// Mitsubishi GX Works2 project: plc   PLC: Q06UDV

PROGRAM MAIN
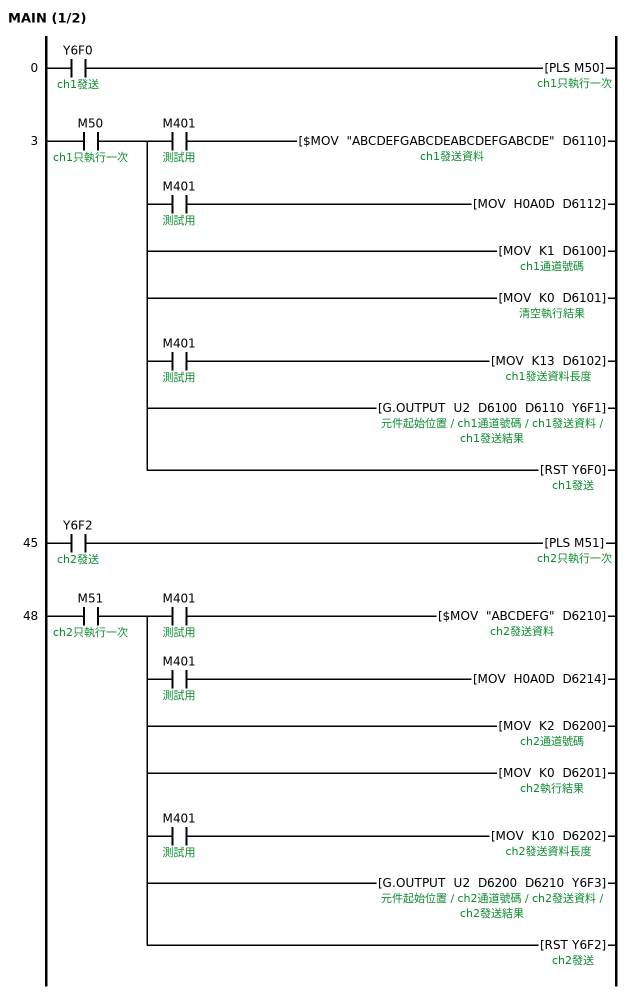
0     LD      Y6F0  ; ch1發送
      PLS     M50  ; ch1只執行一次
3     LD      M50  ; ch1只執行一次
      MPS
      AND     M401  ; 測試用
      $MOV    "ABCDEFGABCDEABCDEFGABCDE" D6110  ; ch1發送資料
      MRD
      AND     M401  ; 測試用
      MOV     H0A0D D6112
      MPP
      MOV     K1 D6100  ; ch1通道號碼
      MOV     K0 D6101  ; 清空執行結果
      MPS
      AND     M401  ; 測試用
      MOV     K13 D6102  ; ch1發送資料長度
      MPP
      G.OUTPUT U2 D6100 D6110 Y6F1  ; 元件起始位置 / ch1發送結果
      RST     Y6F0  ; ch1發送
45    LD      Y6F2  ; ch2發送
      PLS     M51  ; ch2只執行一次
48    LD      M51  ; ch2只執行一次
      MPS
      AND     M401  ; 測試用
      $MOV    "ABCDEFG" D6210  ; ch2發送資料
      MRD
      AND     M401  ; 測試用
      MOV     H0A0D D6214
      MPP
      MOV     K2 D6200  ; ch2通道號碼
      MOV     K0 D6201  ; ch2執行結果
      MPS
      AND     M401  ; 測試用
      MOV     K10 D6202  ; ch2發送資料長度
      MPP
      G.OUTPUT U2 D6200 D6210 Y6F3  ; ch2發送結果
      RST     Y6F2  ; ch2發送
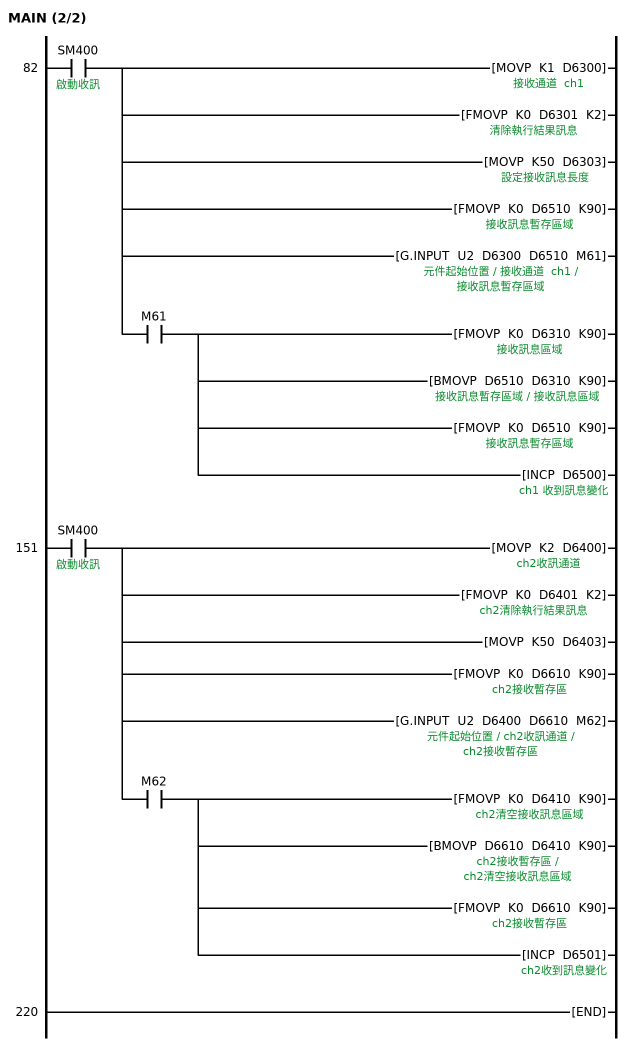
82    LD      SM400  ; 啟動收訊
      MOVP    K1 D6300  ; 接收通道  ch1
      FMOVP   K0 D6301 K2  ; 清除執行結果訊息
      MOVP    K50 D6303  ; 設定接收訊息長度
      FMOVP   K0 D6510 K90  ; 接收訊息暫存區域
      G.INPUT U2 D6300 D6510 M61
      AND     M61
      FMOVP   K0 D6310 K90  ; 接收訊息區域
        [note] 清空接收區
      BMOVP   D6510 D6310 K90
        [note] 從暫存區讀取訊息
      FMOVP   K0 D6510 K90
        [note] 清空暫存區
      INCP    D6500  ; ch1 收到訊息變化
151   LD      SM400  ; 啟動收訊
      MOVP    K2 D6400  ; ch2收訊通道
      FMOVP   K0 D6401 K2  ; ch2清除執行結果訊息
      MOVP    K50 D6403
      FMOVP   K0 D6610 K90  ; ch2接收暫存區
      G.INPUT U2 D6400 D6610 M62
      AND     M62
      FMOVP   K0 D6410 K90  ; ch2清空接收訊息區域
        [note] 清空接收區
      BMOVP   D6610 D6410 K90
        [note] 從暫存區讀取訊息
      FMOVP   K0 D6610 K90
        [note] 清空暫存區
      INCP    D6501  ; ch2收到訊息變化
220   END
END_PROGRAM
